Staubli VAL3: frame.pjx

--- frame.pjx ---
Parameters version=s7.6.1 stackSize=5000 millimeterUnit=true
Program file=buildList.pgx
Program file=checkPoint.pgx
Program file=listAdd.pgx
Program file=loadPage.pgx
Program file=main.pgx
Program file=onBackEvent.pgx
Program file=onEnterEvent.pgx
Program file=onExit.pgx
Program file=onF1Event.pgx
Program file=onF2Event.pgx
Program file=onF3Event.pgx
Program file=onF4Event.pgx
Program file=onF5Event.pgx
Program file=onF6Event.pgx
Program file=onF7Event.pgx
Program file=onF8Event.pgx
Program file=onStart.pgx
Program file=page_changeTrsf.pgx
Program file=refresh.pgx
Program file=refreshDynamic.pgx
Program file=refreshStatic.pgx
Program file=setPointFrame.pgx
Program file=showStatus.pgx
Data file=frame.dtx
Library alias=page path=Disk://kernel/template/page/page.pjx
Library alias=use path=Disk://kernel/userPage/userPage.pjx
Library alias=language path=Disk://kernel/language/language.pjx
Library alias=saveData path=Disk://saveData/saveData.pjx
Library alias=cycleStatus path=Disk://cycleStatus/cycleStatus.pjx
Library alias=tcp path=Disk://kernel/tool/tool.pjx
Type name=FrameItem path=Disk://kernel/template/FrameItem/FrameItem.pjx
Type name=ToolItem path=Disk://kernel/template/ToolItem/ToolItem.pjx

--- frame.dtx ---
num nClockStatus = 835.53
num nFrame = -1
num nKey = -1
num nRefresh = 59941.087
num nTime = 1
num nView
string sEvent = " 0 World"
public string sItems
string sList[11]
  [0] = " 0 World"
  [1] = " 1 frComparateur"
  [2] = " 2 frPiece"
  [3] = " 3 frame3"
  [4] = " 4 frame4"
  [5] = " 5 frame5"
  [6] = " 6 frame6"
  [7] = " 7 frame7"
  [8] = " 8 frame8"
  [9] = " 9 rd"
  [10] = "10 titi"
string sMenu[8]
  [0] = "Teach"
  [1] = "Tool"
  [2] = "Execute"
  [3] = "ALIGN"
  [4] = "Compute"
  [5] = "Mark"
  [6] = "Paste"
  [7] = "Save"
string sMessage
bool bButton[8]
  [0] = true
  [1] = true
  [2] = true
  [3] = true
  [4] = true
  [5] = true
  [6] = true
  [7] = true
bool bLarge
bool bShowStatus
bool bTrigger
frame fSetFrame = {fatherId=world[0]}
pointRx pCheck = {fatherId=world[0]}
pointRx points[3]
  [0] = {fatherId=world[0]}
  [1] = {fatherId=world[0]}
  [2] = {fatherId=world[0]}
mdesc nom_speed = {tmax=100, rmax=100, blend=off}
mdesc nom_speed_2 = {tmax=1, rmax=1, blend=off}
tool tTool = {fatherId=flange[0], ioLink=valve1}

--- main.pgx ---
public program main()
begin
  // INIT
  call onStart()
  // LOOP UNTIL nKey=255
  do
    call refresh()
    nKey=getKey()
    call use:listevent(nKey,nFrame,sEvent)
    nView=use:nView
    switch nKey
      case 259
        // TAB
        bLarge=!bLarge
        call use:setView(bLarge)
      break
      case 263
        call onBackEvent()
      break
      case 271
        call onF1Event()
      break
      case 272
        call onF2Event()
      break
      case 273
        call onF3Event()
      break
      case 274
        call onF4Event()
      break
      case 275
        call onF5Event()
      break
      case 276
        call onF6Event()
      break
      case 277
        call onF7Event()
      break
      case 278
        call onF8Event()
      break
      case 270
        call onEnterEvent()
      break
    endSwitch
    // release the resource
    delay(0)
  until nKey==255
  // on Exit
  call onExit()
end

--- buildList.pgx ---
program buildList()
  local num l_nSize
  local string l_sEvent
  local num i
  local string l_sEmpty
begin
  // INIT the list
  l_sEmpty=""
  call use:stringCopy(l_sEmpty,sList)
  // Build the list
  for i=0 to size(saveData:fFrameItem)-1
    call listAdd(toString("2",i)+" "+saveData:fFrameItem[i].sName)
  endFor
end

--- checkPoint.pgx ---
public program checkPoint(point x_PointToGo, point x_PointStart, bool& x_bUnreached[], tool x_tTool, bool x_bLinear)
  local joint jpO_frameint
  local string message
  local num i
begin
  // check if the pO_frameint is null???
  if (cycleStatus:bCycle==false and cycleStatus:bSimulation==false) or !x_bLinear
    x_bUnreached=(position(x_PointToGo,world)=={0,0,0,0,0,0})
    //
    if !x_bUnreached
      //
      // look if the pO_frameint that you want to reach is valid
      if x_bLinear
        //
        // use the percentage....
        //
        for i=0.1 to 1 step 0.1
          pCheck.trsf=interpolateL(position(x_PointStart,world),position(x_PointToGo,world),i)
          x_bUnreached=!pointToJoint(x_tTool,herej(),pCheck,jpO_frameint)
          if x_bUnreached
            return
          endIf
        endFor
      else
        // joint move or check only the working area
        x_PointToGo.config={sfree,efree,wfree}
        x_bUnreached=!pointToJoint(x_tTool,herej(),x_PointToGo,jpO_frameint)
      endIf
    endIf
  endIf
end

--- listAdd.pgx ---
program listAdd(string x_sEvent)
begin
  // add in the queue
  if sList!=""
    insert(sList[size(sList)])
  endIf
  sList[size(sList)-1]=x_sEvent
end

--- loadPage.pgx ---
program loadPage(string x_sPage, string& x_sItems[])
// load the next page
  local num i
begin
  // look if the page libload is correct
  i=page:libLoad(x_sPage)
  delay(0)
  logMsg("[VALPLAST] INTERFACE:PAGE LIBLOAD "+x_sPage+" result "+toString("",i))
  if i!=0
    popUpMsg("Loading page "+x_sPage+" error CODE "+toString("",i))
  else
    // copy all the field from x_sItems to the next page
    call use:stringCopy(x_sItems,page:sItems)
    call page:main()
    // to give back
    call use:stringCopy(page:sItems,x_sItems)
  endIf
end

--- onBackEvent.pgx ---
program onBackEvent()
  local string l_sItem
  local num i
begin
  //
  // rename
  //
  if nFrame>0
    l_sItem=saveData:fFrameItem[nFrame].sName
    if l_sItem!=""
      i=find(sEvent,l_sItem)
    else
      i=len(toString("",nFrame))+3
    endIf
    if i!=-1
      // clean the line
      call use:listcursor(use:nView,false)
      // read the name
      call use:read(40-use:nBottomX+i-1,nView+1,l_sItem,10,false)
      saveData:fFrameItem[nFrame].sName=l_sItem
      call buildList()
      use:bUseRefresh=true
    endIf
  endIf
end

--- onEnterEvent.pgx ---
program onEnterEvent()
begin
  //
  // Change the frame coordinate
  //
  if nFrame>0
    call page_changeTrsf(saveData:fFrameItem[nFrame].fFrame.trsf,false,false,sEvent,"")
  endIf
end

--- onExit.pgx ---
program onExit()
begin
  // save it
  saveData:libSave()
  use:bUseRefresh=true
end

--- onF1Event.pgx ---
program onF1Event()
  local num l_nFrame
  local string l_sEvent
begin
  // look if the bButton is enable
  if bButton[0] and nFrame>0
    // teach the frame
    call setPointFrame(saveData:fFrameItem[nFrame].fFrame.trsf,nFrame)
    // release
    call use:nullKey(nKey)
    use:bUseRefresh=true
  endIf
end

--- onF2Event.pgx ---
program onF2Event()
  local string l_sEmpty
begin
  // look if the bButton is enable
  if bButton[1]
    // tool selection
    call loadPage("Disk://kernel/page/tool",l_sEmpty)
    //
    saveData:nFrameTool=saveData:nIndexTool
  endIf
end

--- onF3Event.pgx ---
program onF3Event()
  local tool l_tTool
begin
  // look if the bButton is enable
  if bButton[2]
    //
    // get the tool
    call tcp:getTool(tTool,saveData:nFrameTool)
    if nFrame>0
      call use:timerDialog("Frame "+sEvent+" actived",3)
      fSetFrame.trsf=saveData:fFrameItem[nFrame].fFrame.trsf
    else
      call use:timerDialog("WORLD Frame actived",3)
      fSetFrame=world
    endIf
    $jogContext(tTool,fSetFrame,0)
    // save the  actual frame
    saveData:nFrameActive=nFrame
  endIf
end

--- onF4Event.pgx ---
program onF4Event()
  local point l_pPoint
begin
  // look if the bButton is enable
  if bButton[3]
    // get the tool
    call tcp:getTool(tTool,saveData:nFrameTool)
    l_pPoint=here(tTool,world)
    l_pPoint.trsf=align(l_pPoint.trsf,fSetFrame.trsf)
    movej(l_pPoint,tTool,nom_speed)
    call use:timerDialog(" ALIGN.... ",1)
    watch(isEmpty() or isKeyPressed(255),3)
    if !isEmpty()
      resetMotion()
    endIf
    delay(2)
  endIf
end

--- onF5Event.pgx ---
program onF5Event()
  local trsf l_trOffset
  local string l_sButton[2]
  local bool l_bResult
  local trsf l_trResult
  local string l_sMessage
begin
  // look if the bButton is enable
  if bButton[4]
    if nFrame>0
      // compute using a trsf
      call page_changeTrsf(l_trOffset,false,false,"COMPUTE","")
      l_sMessage=" use this frame...#"
      l_sMessage=l_sMessage+toString("",saveData:fFrameItem[nFrame].fFrame.trsf.x)+","+toString("",saveData:fFrameItem[nFrame].fFrame.trsf.y)+","+toString("",saveData:fFrameItem[nFrame].fFrame.trsf.z)
      l_sMessage=l_sMessage+","+toString("",saveData:fFrameItem[nFrame].fFrame.trsf.rx)+","+toString("",saveData:fFrameItem[nFrame].fFrame.trsf.ry)+","+toString("",saveData:fFrameItem[nFrame].fFrame.trsf.rz)
      l_sMessage=l_sMessage+"#"+toString("",l_trOffset.x)+","+toString("",l_trOffset.y)+","+toString("",l_trOffset.z)+","+toString("",l_trOffset.rx)+","+toString("",l_trOffset.ry)+","+toString("",l_trOffset.rz)
      l_trResult=saveData:fFrameItem[nFrame].fFrame.trsf*l_trOffset
      l_sMessage=l_sMessage+"##"+toString("",l_trResult.x)+","+toString("",l_trResult.y)+","+toString("",l_trResult.z)+","+toString("",l_trResult.rx)+","+toString("",l_trResult.ry)+","+toString("",l_trResult.rz)
      call language:getYesNo(l_sButton)
      call use:yes_no(l_sMessage,l_sButton,l_bResult)
      // check if is ok
      if l_bResult
        saveData:fFrameItem[nFrame].fFrame.trsf=l_trResult
      endIf
    endIf
  endIf
end

--- onF6Event.pgx ---
program onF6Event()
  local num i
  local string l_sItem
begin
  // look if the bButton is enable
  if bButton[5]
    // mark
    // deselect all
    for i=0 to size(sList)-1
      if find(sList[i],"#")!=-1
        sList[i]=right(sList[i],len(sList[i])-1)
      endIf
    endFor
    // select it
    sList[nFrame]="#"+sList[nFrame]
    nFrame=nFrame+1
    use:nView=use:nView+1
  endIf
end

--- onF7Event.pgx ---
program onF7Event()
  local num i
  local num l_nFrame
begin
  // look if the bButton is enable
  if bButton[6]
    // paste it
    l_nFrame=-1
    for i=0 to size(sList)-1
      if find(sList[i],"#")!=-1
        l_nFrame=i
      endIf
    endFor
    if l_nFrame!=-1
      // paste it
      if l_nFrame==0
        saveData:fFrameItem[nFrame].fFrame.trsf={0,0,0,0,0,0}
      else
        saveData:fFrameItem[nFrame].pO.trsf=saveData:fFrameItem[l_nFrame].pO.trsf
        saveData:fFrameItem[nFrame].pX.trsf=saveData:fFrameItem[l_nFrame].pX.trsf
        saveData:fFrameItem[nFrame].pY.trsf=saveData:fFrameItem[l_nFrame].pY.trsf
        saveData:fFrameItem[nFrame].fFrame.trsf=saveData:fFrameItem[l_nFrame].fFrame.trsf
      endIf
      call use:timerDialog("PASTE FRAME "+toString("",l_nFrame)+" to FRAME "+toString("",nFrame),3)
    endIf
  endIf
end

--- onF8Event.pgx ---
program onF8Event()
  local string l_sMessage
begin
  // look if the bButton is enable
  if bButton[7]
    // none ...
  endIf
end

--- onStart.pgx ---
program onStart()
  local num i
  local string l_sMessage
begin
  // logMsg
  logMsg("[VALPLAST] INTERFACE:PAGE...")
  // be aware these value will change all the value
  call language:message(l_sMessage,129)
  popUpMsg(l_sMessage)
  // reset the Key pressure
  call use:nullKey(nKey)
  // define the list
  call buildList()
  // build the page
  call refreshStatic()
  // define the list
end

--- page_changeTrsf.pgx ---
public program page_changeTrsf(trsf& x_tTrsf[], bool x_bUseFrame, bool x_bUseReset, string x_sTitle, string x_sComment)
  local string l_sEvent
  local num l_nFrame
  local num l_nView
  local bool l_bRefresh
  local bool l_bTest
  local num l_nKey
  local num i
  local string l_sMessage
  local trsf l_tTrsf
  local string l_sItem
  local string l_sEmpty
begin
  logMsg("[KERNEL] INTERFACE:PAGE changeTrsf "+x_sTitle)
  l_bRefresh=false
  l_nFrame=0
  l_nView=0
  call use:setSizeList(19,0,19,8)
  call use:setView(false)
  l_tTrsf=x_tTrsf
  //
  do
    cls()
    call use:type(0,12,x_sComment)
    call use:typeMenu(8,"OK")
    if x_bUseReset
      call language:message(l_sMessage,184)
      call use:strfill(l_sMessage,5,l_sMessage)
      call use:type(21,13,l_sMessage)
    endIf
    call use:listcreate(x_sTitle)
    l_sItem="coord  X > "+toString(".3",l_tTrsf.x)
    call use:listadd(l_sItem)
    l_sItem="coord  Y > "+toString(".3",l_tTrsf.y)
    call use:listadd(l_sItem)
    l_sItem="coord  Z > "+toString(".3",l_tTrsf.z)
    call use:listadd(l_sItem)
    l_sItem="coord RX > "+toString(".3",l_tTrsf.rx)
    call use:listadd(l_sItem)
    l_sItem="coord RY > "+toString(".3",l_tTrsf.ry)
    call use:listadd(l_sItem)
    l_sItem="coord RZ > "+toString(".3",l_tTrsf.rz)
    call use:listadd(l_sItem)
    use:nView=l_nFrame
    call use:listupdate(l_nFrame-l_nView)
    do
      l_nView=use:nView
      l_nKey=get()
      call use:listevent(l_nKey,l_nFrame,l_sEvent)
      switch l_nKey
        case 270
          //
          // clean the line
          call use:listcursor(use:nView,false)
          switch l_nFrame
            case 0
              //  x-value
              call use:changeValue(l_tTrsf.x,0,0,10+40-use:nBottomX,use:nView+1,l_sEmpty)
            break
            case 1
              //  y-value
              call use:changeValue(l_tTrsf.y,0,0,10+40-use:nBottomX,use:nView+1,l_sEmpty)
            break
            case 2
              //  z-value
              call use:changeValue(l_tTrsf.z,0,0,10+40-use:nBottomX,use:nView+1,l_sEmpty)
            break
            case 3
              //  rx-value
              call use:changeValue(l_tTrsf.rx,0,0,10+40-use:nBottomX,use:nView+1,l_sEmpty)
            break
            case 4
              //  ry-value
              call use:changeValue(l_tTrsf.ry,0,0,10+40-use:nBottomX,use:nView+1,l_sEmpty)
            break
            case 5
              //  rz-value
              call use:changeValue(l_tTrsf.rz,0,0,10+40-use:nBottomX,use:nView+1,l_sEmpty)
            break
          endSwitch
          l_bRefresh=true
        break
        case 278
          // VALIDATE
          x_tTrsf=l_tTrsf
        break
        case 275
          // RESET
          if x_bUseReset
            l_tTrsf={0,0,0,0,0,0}
            l_bRefresh=true
          endIf
        break
      endSwitch
    until l_bRefresh==true or l_nKey==255 or l_nKey==278
    l_bRefresh=false
  until l_nKey==255 or l_nKey==278
  // release the resource
  call use:nullKey(l_nKey)
  if !cycleStatus:bCycle and !cycleStatus:bSimulation
    resetMotion()
  endIf
end

--- refresh.pgx ---
program refresh()
// // page refresh
begin
  // refresh the static message
  if !bShowStatus
    if (nKey>=270 and nKey<=278) or use:bUseRefresh
      call refreshStatic()
      call refreshDynamic()
    else
      if !bShowStatus
        // refresh the Dynamic message
        if (clock()-nRefresh>nTime)
          call refreshDynamic()
        endIf
      endIf
    endIf
  endIf
  // show the coordinate
  call showStatus()
  // release the resource
  delay(0)
end

--- refreshStatic.pgx ---
program refreshStatic()
  local string l_sMenu
  local string l_sMessage
  local string l_sName
begin
  cls()
  //
  // set the view of the page..
  //
  // SET THE PAGE NUMBER
  use:nPage=150
  // USE <>PROFILE for <>PAGE
  use:nPage=use:nPage+abs(limit(saveData:mode,0,2)-2)
  // SET THE VIEW OF THE PAGE
  call language:page(l_sMenu,use:nPage)
  // define the menu
  call use:stringToArray(l_sMenu,sMenu)
  call use:setMenu(sMenu,true,3)
  call use:getMenu(sMenu,bButton)
  //
  // CREATE THE LIST
  //
  // define your list size for default
  call use:setSizeList(20,0,18,11)
  call use:setView(bLarge)
  //
  call use:listcreate("")
  //
  call use:listadd(sList)
  //
  // refresh the cursor
  use:nView=nView
  // refresh the list
  call use:listupdate(0)
  // show the tool
  call language:message(l_sMessage,124)
  call tcp:getName(l_sName,saveData:nFrameTool)
  call use:type(0,0,l_sMessage+">"+toString("",saveData:nFrameTool)+" "+saveData:tData[saveData:nFrameTool].name)
  // show the frame
  call use:type(0,1,"Frame>"+toString("",saveData:nFrameActive)+" "+saveData:fFrameItem[saveData:nFrameActive].sName)
end

--- setPointFrame.pgx ---
program setPointFrame(trsf& x_trsfFrame[], num x_nFrame)
  local string l_sMessage[2]
  local num l_nStep
  local string l_sButton[8]
  local num l_nResult
  local tool l_tTool
  local num i
  local point l_pHere
  local bool l_bUnreachable
  local string l_sTcp
begin
  //
  //  Change the Frame associate to the Trajectory
  //
  cls()
  l_nStep=0
  l_sButton[0]=">>"
  l_sButton[1]="<<"
  //
  // copY_frame from saveData
  //
  points[0].trsf=saveData:fFrameItem[x_nFrame].pO.trsf
  points[1].trsf=saveData:fFrameItem[x_nFrame].pX.trsf
  points[2].trsf=saveData:fFrameItem[x_nFrame].pY.trsf
  //
  call language:message(l_sMessage,167)
  l_sButton[6]=l_sMessage
  //
  call language:message(l_sMessage,150)
  l_sButton[7]=l_sMessage
  call saveData:getTool(l_tTool,saveData:nFrameTool)
  //
  while l_nStep<10
    //
    //
    resetMotion()
    l_pHere=here(l_tTool,world)
    //
    switch l_nStep
      case -1
        return
      break
      case 0
        // take the Origin
        call checkPoint(points[0],points[0],l_bUnreachable,l_tTool,false)
        //
        call language:message(l_sMessage,194)
        call language:message(l_sMessage[1],168)
        l_sMessage=l_sMessage+"#"+l_sMessage[1]
        if !l_bUnreachable and cycleStatus:nWorkingMode==1
          call language:message(l_sMessage[1],203)
          l_sMessage=l_sMessage+"#"+l_sMessage[1]
          //
          movej(points[0],l_tTool,nom_speed)
        endIf
        call use:questionDialog(l_sMessage,l_sButton,l_nResult)
        if l_nResult==8
          points[0]=here(l_tTool,world)
          call language:message(l_sMessage,193)
          call use:type(2,11,l_sMessage)
        else
          if l_nResult==7
            call language:message(l_sMessage,198)
            call page_changeTrsf(points[0].trsf,false,false,l_sMessage,"")
          else
            call use:clear(0,11)
          endIf
        endIf
      break
      case 1
        //take the X pO_frameint
        call checkPoint(points[1],l_pHere,l_bUnreachable,l_tTool,true)
        //
        call language:message(l_sMessage,195)
        call language:message(l_sMessage[1],168)
        l_sMessage=l_sMessage+"#"+l_sMessage[1]
        if !l_bUnreachable and cycleStatus:nWorkingMode==1
          call language:message(l_sMessage[1],203)
          l_sMessage=l_sMessage+"#"+l_sMessage[1]
          //
          movel(points[1],l_tTool,nom_speed)
        endIf
        call use:questionDialog(l_sMessage,l_sButton,l_nResult)
        if l_nResult==8
          points[1]=here(l_tTool,world)
          call language:message(l_sMessage,193)
          call use:type(2,11,l_sMessage)
        else
          if l_nResult==7
            call language:message(l_sMessage,199)
            call page_changeTrsf(points[1].trsf,false,false,l_sMessage+" X","")
          else
            call use:clear(0,11)
          endIf
        endIf
      break
      case 2
        // take the Y pO_frameint
        call checkPoint(points[2],l_pHere,l_bUnreachable,l_tTool,true)
        //
        call language:message(l_sMessage,196)
        call language:message(l_sMessage[1],168)
        l_sMessage=l_sMessage+"#"+l_sMessage[1]
        call language:message(l_sMessage[1],203)
        if !l_bUnreachable and cycleStatus:nWorkingMode==1
          call language:message(l_sMessage[1],203)
          l_sMessage=l_sMessage+"#"+l_sMessage[1]
          //
          movel(points[2],l_tTool,nom_speed)
        endIf
        call use:questionDialog(l_sMessage,l_sButton,l_nResult)
        if l_nResult==8
          points[2]=here(l_tTool,world)
          call language:message(l_sMessage,193)
          call use:type(2,11,l_sMessage)
        else
          if l_nResult==7
            call language:message(l_sMessage,199)
            call page_changeTrsf(points[2].trsf,false,false,l_sMessage+" Y","")
          else
            call use:clear(0,11)
          endIf
        endIf
      break
      case 3
        // set the frame
        if setFrame(points[0],points[1],points[2],fSetFrame)==0
          x_trsfFrame=fSetFrame.trsf
          // copY_frame back to save DATA
          saveData:fFrameItem[x_nFrame].pO.trsf=points[0].trsf
          saveData:fFrameItem[x_nFrame].pX.trsf=points[1].trsf
          saveData:fFrameItem[x_nFrame].pY.trsf=points[2].trsf
          //
        else
          call language:message(l_sMessage,183)
          popUpMsg(l_sMessage+toString("",setFrame(points[0],points[1],points[2],fSetFrame)))
        endIf
        return
      break
      //
    endSwitch
    // step control
    if l_nResult==0 or l_nResult==1
      l_nStep=l_nStep+1
      cls()
      delay(0)
    else
      if l_nResult==2
        l_nStep=l_nStep-1
      else
        if l_nResult==-1
          return
        endIf
      endIf
    endIf
  endWhile
end

--- showStatus.pgx ---
program showStatus()
  local joint l_jHere
  local point l_pHere
  local string l_sMessage[2]
  local tool l_tTool
begin
  //
  // show an dialog box with
  // the current Joint/cartesian position
  //
  call tcp:getTool(l_tTool,saveData:nFrameTool)
  if cycleStatus:nWorkingStatus>1 and cycleStatus:nWorkingStatus<5 and cycleStatus:nWorkingMode==1
    // set a timer of x second then the message disappear ..
    if !bTrigger
      nClockStatus=clock()
      bTrigger=true
      bShowStatus=true
    endIf
    if clock()-nClockStatus<saveData:nTimeDialog
      if cycleStatus:nWorkingStatus==2
        l_jHere=herej()
        l_sMessage="J1:"+toString("7.1",l_jHere.j1)
        l_sMessage=l_sMessage+"  J2:"+toString("7.1",l_jHere.j2)
        l_sMessage=l_sMessage+"  J3:"+toString("7.1",l_jHere.j3)+"#"
        l_sMessage=l_sMessage+"J4:"+toString("7.1",l_jHere.j4)
        l_sMessage=l_sMessage+"  J5:"+toString("7.1",l_jHere.j5)
        l_sMessage=l_sMessage+"  J6:"+toString("7.1",l_jHere.j6)
      else
        l_pHere=here(l_tTool,fSetFrame)
        l_sMessage="X :"+toString("7.1",l_pHere.trsf.x)
        l_sMessage=l_sMessage+"  Y :"+toString("7.1",l_pHere.trsf.y)
        l_sMessage=l_sMessage+"  Z :"+toString("7.1",l_pHere.trsf.z)+"#"
        l_sMessage=l_sMessage+"RX:"+toString("7.1",l_pHere.trsf.rx)
        l_sMessage=l_sMessage+"  RY:"+toString("7.1",l_pHere.trsf.ry)
        l_sMessage=l_sMessage+"  RZ:"+toString("7.1",l_pHere.trsf.rz)
      endIf
      call use:timerDialog(l_sMessage,3)
    else
      // disable it
      bShowStatus=false
      bTrigger=false
    endIf
  else
    // reset it
    if bTrigger
      resetMotion()
    endIf
    bTrigger=false
    bShowStatus=false
  endIf
end
